// TIA Portal V19 export
TYPE "UDT_SIM_MTR"
   STRUCT
      simFb : Bool;
      simCtrl : Bool;
   END_STRUCT;
END_TYPE
